PROGRAM KUKA_IO
VAR_INPUT
	LogText : STRING;
END_VAR

KR1();
KR2();
KR3();
KR4();
KR5();

END_PROGRAM

(* stored: Version 1.1.0.1, ProductVersion 3.1.4024.12
   POU KUKA_IO: Id {8ae2eb55-87e1-4ea9-a7b9-09ebadc6d917}, SpecialFunc None *)
